// TIA Portal V19 export
TYPE "type_XyzToU3"
// stored: Access Published, Namespace Unit3
   STRUCT
      requeset : "Unit3.type_xyzRequestData";
      response : "Unit3.type_xyzResponsetData";
   END_STRUCT;
END_TYPE
